// TwinCAT 3 PLC project EtherCATStateControl
// ProgramVersion: 3.1.4024.0
// libraries:
//   Tc2_EtherCAT, * (Beckhoff Automation GmbH)
//   Tc2_Standard, * (Beckhoff Automation GmbH)
//   Tc2_System, * (Beckhoff Automation GmbH)
//   Tc3_Module, * (Beckhoff Automation GmbH)
// project tree:
//   / PlcTask.TcTTO
//   POUs/ FB_SetSlaveState.TcPOU, ITF_SetSlaveState.TcIO, MAIN.TcPOU
// real-time tasks:
//   TASK PlcTask: cycle T#10ms, priority 20, ADS port 350
// I/O:
//   DEVICE Device 1 (EtherCAT), AmsNetId 192.168.5.28.2.1
//     Term 1 (EK1100) [EK1100 EtherCAT Coupler (2A E-Bus)]
//       Term 2 (EL6652) [EL6652 EtherNet/IP Scanner (Master)]
//   DEVICE Device 2 (ECAT EIP Scanner (EL6652)), AmsNetId 192.168.5.28.3.1
//     Box 3 (EtherNet/IP Slave (generic)) // <INFO> </INFO> <EDS> C:\TwinCAT\3.1\Config\Io\EtherNetIP\ </EDS>
// variable links:
//   EtherCATStateControl Instance <-> Device 1 (EtherCAT)/Term 1 (EK1100)/Term 2 (EL6652)
//     PlcTask Inputs/MAIN.fbDeviceStateCtrl.nSlaveAddr <-> InfoData/AdsAddr/port
//     PlcTask Inputs/MAIN.fbDeviceStateCtrl.sAMSNet <-> InfoData/AdsAddr/netId
//   EtherCATStateControl Instance <-> Device 2 (ECAT EIP Scanner (EL6652))/Box 3 (EtherNet/IP Slave (generic))
//     PlcTask Inputs/MAIN.EIPDataIn <-> Connection 1 (Input/Output)/Inputs/MAIN.EIPDataIn
//     PlcTask Inputs/MAIN.EIPDataIn @bit {16..64 step 16} <-> Connection 1 (Input/Output)/Inputs/Var {25..28}  (4 links)
//     PlcTask Outputs/MAIN.EIPDataOut <-> Connection 1 (Input/Output)/Outputs/MAIN.EIPDataOut
//     PlcTask Outputs/MAIN.EIPDataOut @bit 16 <-> Connection 1 (Input/Output)/Outputs/Var 23
//     PlcTask Outputs/MAIN.EIPDataOut @bit 32 <-> Connection 1 (Input/Output)/Outputs/Var 42
//     PlcTask Outputs/MAIN.EIPDataOut @bit 48 <-> Connection 1 (Input/Output)/Outputs/Var 43
//     PlcTask Outputs/MAIN.EIPDataOut @bit 64 <-> Connection 1 (Input/Output)/Outputs/Var 44

CONFIGURATION EtherCATStateControl
    RESOURCE PLC ON TwinCAT3
        TASK PlcTask(INTERVAL := T#10ms, PRIORITY := 20);
        PROGRAM MAIN WITH PlcTask : MAIN;
    END_RESOURCE
END_CONFIGURATION

// ---- POUs/ITF_SetSlaveState.TcIO
INTERFACE ITF_SetSlaveState

PROPERTY CurrentState : ST_EcSlaveState
GET
END_GET
END_PROPERTY

METHOD GetState : BOOL
VAR_INPUT
	tTimeout   						: TIME := T#10S; // Timeout time for ECSetSlaveState FB
END_VAR
END_METHOD

METHOD ResetStateToOp : BOOL
VAR_INPUT
	tTimeout   						: TIME := T#10S; // Timeout time for ECSetSlaveState FB
END_VAR
END_METHOD

METHOD SetState : BOOL
VAR_INPUT
	reqState   						: WORD; // Holds the state the device will be set to 1 = Init, 2 = PreOP, 3 =  Bootstrap, 4 = SafeOp, 8 = OP
    tTimeout   						: TIME := T#10S; // Timeout time for ECSetSlaveState FB
END_VAR
END_METHOD

END_INTERFACE

// ---- POUs/MAIN.TcPOU
PROGRAM MAIN
VAR
	fbDeviceStateCtrl		: FB_SetSlaveState;
	_bSetToInit				: BOOL;
	_bSetToOP				: BOOL;
	_bResetToOp				: BOOL;
	
	EIPDataIn AT %I*		: ARRAY[1..5] OF WORD; 
	EIPDataOut AT %Q*		: ARRAY[1..5] OF WORD; 

END_VAR

IF _bSetToInit THEN
	IF fbDeviceStateCtrl.SetState(1,T#2S) THEN
		_bSetToInit := FALSE;
	END_IF
END_IF

IF _bSetToOP THEN
	IF fbDeviceStateCtrl.SetState(8, T#2S) THEN
		_bSetToOP := FALSE;
	END_IF
END_IF

IF _bResetToOp THEN
	IF fbDeviceStateCtrl.ResetStateToOp(T#3S) THEN
		_bResetToOp := FALSE;
	END_IF
END_IF

END_PROGRAM

// ---- POUs/FB_SetSlaveState.TcPOU
(*
:Description: FUNCTION block to control EtherCAT slave device state machine

:Instructions for use: Requires Tc2_EtherCAT Library

Version history:

+-------------+------------+----------------+----------+------------------------------------------+
|Date         | Version    | created under  | Author   | Remark                                   |
+=============+============+================+==========+==========================================+
|2024-12-12   | 1.0.0.0    | 			    | G.P      | Draft					                  |
+-------------+------------+----------------+----------+------------------------------------------+
|			  | 		   | 			    | 		   | Release							      |
+-------------+------------+----------------+----------+------------------------------------------+

*)
FUNCTION_BLOCK FB_SetSlaveState IMPLEMENTS ITF_SetSlaveState
VAR_INPUT
	sAMSNet		  AT %I*			: AMSNETID; // Linked to EtherCAT master
    nSlaveAddr    AT %I*     		: UINT;	    //  Linked to PortID of slave device
END_VAR
VAR_OUTPUT
END_VAR
VAR
	fbSetECSlaveState				: Tc2_EtherCAT.FB_EcSetSlaveState;
	fbGetECSlaveState				: Tc2_EtherCAT.FB_EcGetSlaveState;
	_nState							: UINT;
    _sNetId       					: T_AmsNetId; // Must have a value
	_CurrentState					: ST_EcSlaveState;
END_VAR

PROPERTY CurrentState : ST_EcSlaveState
GET
CurrentState := _CurrentState;
END_GET
END_PROPERTY

METHOD GetState : BOOL
VAR_INPUT
	tTimeout   						: TIME := T#10S; // Timeout time for ECSetSlaveState FB
END_VAR
GetState := FALSE;
CASE _nState OF
0:
   _sNetID := F_CreateAmsNetId( sAMSNet ); // Convert linked EtherCAT Master AMS address and convert to string format FB's can use.
   _nState := 1;

1:
  
	// Get slave current state so we can check it changed to the requested state
	fbGetECSlaveState(
		sNetId:= _sNetId , 
		nSlaveAddr:= nSlaveAddr, 
		bExecute:= TRUE, 
		tTimeout:= tTimeout);
		_nState := 2; // Goto next state
  
2:  
	fbGetECSlaveState(bExecute := FALSE, state=> _CurrentState ); // Reset the execute flag of get slave state
	// Check get slave state has completed without errors
	IF (NOT fbGetECSlaveState.bBusy) AND (NOT fbGetECSlaveState.bError) THEN
		_nState := 3; // Move on
	END_IF
3:
   // All complete so reset flags
   GetState := TRUE;
   _nState := 0;

100:
   ;                     // Error handling..
END_CASE
END_METHOD

METHOD ResetStateToOp : BOOL
VAR_INPUT
	tTimeout		: TIME := T#10S; // Timeout time for ECSetSlaveState FB
END_VAR
ResetStateToOp := FALSE;
CASE _nState OF
0:
   _sNetID := F_CreateAmsNetId( sAMSNet ); // Convert linked EtherCAT Master AMS address and convert to string format FB's can use.
   _nState := 1;

1:
   // Set the slave to the state requested to goto	
   fbSetECSlaveState(
	sNetId:= _sNetId, 
	nSlaveAddr:= nSlaveAddr, // Linked port  
	bExecute:= TRUE , 
	tTimeout:= tTimeout , 
	reqState:= 1); // State requested to init
    _nState := _nState + 1; // Goto next state
2:
  
  fbSetECSlaveState( bExecute := FALSE); // Reset the execute flag of set slave state
  // Check the set slave state has completed without errors
  IF (NOT fbSetECSlaveState.bBusy) AND (NOT fbSetECSlaveState.bError) THEN
	 // Get slave current state so we can check it changed to the requested state
	 fbGetECSlaveState(
		sNetId:= _sNetId , 
		nSlaveAddr:= nSlaveAddr, 
		bExecute:= TRUE, 
		tTimeout:= tTimeout);
		_nState := 3; // Goto next state
  END_IF
  
  IF fbSetECSlaveState.bError THEN
	  _nState := 100;
  END_IF
  
3:  
	fbGetECSlaveState(bExecute := FALSE, state=> _CurrentState ); // Reset the execute flag of get slave state
	// Check get slave state has completed without errors
	IF (NOT fbGetECSlaveState.bBusy) AND (NOT fbGetECSlaveState.bError) THEN
		_nState := 4; // Move on
	END_IF
	
4:
	// Make sure in correct state
  	IF _CurrentState.deviceState = Tc2_EtherCAT.EC_DEVICE_STATE_INIT THEN
  	   _nState := _nState + 1; // Goto next state
	END_IF;
	
5:
	// Set the slave to the state requested to goto	
   fbSetECSlaveState(
	sNetId:= _sNetId, 
	nSlaveAddr:= nSlaveAddr, // Linked port  
	bExecute:= TRUE , 
	tTimeout:= tTimeout , 
	reqState:= 8); // State requested to OP
    _nState := _nState + 1; // Goto next state
	
6:
	fbSetECSlaveState( bExecute := FALSE); // Reset the execute flag of set slave state
  	// Check the set slave state has completed without errors
  	IF (NOT fbSetECSlaveState.bBusy) AND (NOT fbSetECSlaveState.bError) THEN
		// Get slave current state so we can check it changed to the requested state
	 	fbGetECSlaveState(
			sNetId:= _sNetId , 
			nSlaveAddr:= nSlaveAddr, 
			bExecute:= TRUE, 
			tTimeout:= tTimeout);
			_nState := _nState + 1; // Goto next state
  	END_IF
  
	IF fbSetECSlaveState.bError THEN
		_nState := 100;
  	END_IF
	
7:  
  	fbGetECSlaveState(bExecute := FALSE, state=> _CurrentState ); // Reset the execute flag of get slave state
	// Check get slave state has completed without errors
	IF (NOT fbGetECSlaveState.bBusy) AND (NOT fbGetECSlaveState.bError) THEN
		_nState := _nState + 1; // Goto next state
	END_IF
	
8:
	// Compare requested state with actual state
  	IF _CurrentState.deviceState = Tc2_EtherCAT.EC_DEVICE_STATE_OP THEN
  	    _nState := _nState + 1; // Goto next state
	END_IF;
	
9:
   // All complete so reset flags
   ResetStateToOp := TRUE;
   _nState := 0;

100:
   ;                     // Error handling..
END_CASE
END_METHOD

METHOD SetState : BOOL
VAR_INPUT
	reqState   						: WORD; // Holds the state the device will be set to 1 = Init, 2 = PreOP, 3 =  Bootstrap, 4 = SafeOp, 8 = OP
    tTimeout   						: TIME := T#10S; // Timeout time for ECSetSlaveState FB
END_VAR
SetState := FALSE;
CASE _nState OF
0:
   _sNetID := F_CreateAmsNetId( sAMSNet ); // Convert linked EtherCAT Master AMS address and convert to string format FB's can use.
   _nState := 1;

1:
   // Set the slave to the state requested to goto	
   fbSetECSlaveState(
	sNetId:= _sNetId, 
	nSlaveAddr:= nSlaveAddr, // Linked port  
	bExecute:= TRUE , 
	tTimeout:= tTimeout , 
	reqState:= reqState); // State requested to goto
    _nState := _nState + 1; // Goto next state
2:
  
  fbSetECSlaveState( bExecute := FALSE); // Reset the execute flag of set slave state
  // Check the set slave state has completed without errors
  IF (NOT fbSetECSlaveState.bBusy) AND (NOT fbSetECSlaveState.bError) THEN
	 // Get slave current state so we can check it changed to the requested state
	 fbGetECSlaveState(
		sNetId:= _sNetId , 
		nSlaveAddr:= nSlaveAddr, 
		bExecute:= TRUE, 
		tTimeout:= tTimeout);
		_nState := 3; // Goto next state
  END_IF
  
  IF fbSetECSlaveState.bError THEN
	  _nState := 100;
  END_IF
  
3:  
	fbGetECSlaveState(bExecute := FALSE, state=> _CurrentState ); // Reset the execute flag of get slave state
	// Check get slave state has completed without errors
	IF (NOT fbGetECSlaveState.bBusy) AND (NOT fbGetECSlaveState.bError) THEN
		_nState := 4; // Move on
	END_IF
4:
	// Compare requested state with actual state
	CASE (reqState) OF
		  1:
		  	IF _CurrentState.deviceState = Tc2_EtherCAT.EC_DEVICE_STATE_INIT THEN
		  	    _nState := 5; // Move to completed state
			END_IF;
		  2:
		  	IF _CurrentState.deviceState = Tc2_EtherCAT.EC_DEVICE_STATE_PREOP THEN
		  	    _nState := 5; // Move to completed state
			END_IF;
          4:
		  	IF _CurrentState.deviceState = Tc2_EtherCAT.EC_DEVICE_STATE_SAFEOP THEN
		  	    _nState := 5; // Move to completed state
			END_IF;
		  8:
		  	IF _CurrentState.deviceState = Tc2_EtherCAT.EC_DEVICE_STATE_OP THEN
		  	    _nState := 5; // Move to completed state
			END_IF;
	  END_CASE
5:
   // All complete so reset flags
   SetState := TRUE;
   _nState := 0;

100:
   ;                     // Error handling..
END_CASE
END_METHOD

END_FUNCTION_BLOCK
